TYPE ST_TrailerSection EXTENDS ST_SectionBase :
STRUCT
END_STRUCT
END_TYPE

(* stored: Version 1.1.0.1, ProductVersion 3.1.4024.12
   DUT ST_TrailerSection: Id {64f054fc-b3ff-4f62-a5b2-dfd14112634c} *)
